// TIA Portal V18 export
FUNCTION "HMI screen" : Void   // FC18, LAD
{ S7_Optimized_Access := 'TRUE' }
VERSION : 0.1
// stored: AutoNumber true, IsIECCheckEnabled false, SetENOAutomatically false, UDAEnableTagReadback false
   VAR_TEMP
      temp1 : Bool;
      temp2 : Bool;
      temp3 : Bool;
      temp10 : Bool;
      temp11 : Bool;
      "dearing A" : Bool;
      "dearing A_1" : Bool;
      dearingA : Bool;
   END_VAR
   VAR_TEMP   // added for the SCL form of the ladder/FBD networks
      _w1 : Bool;
      _w2 : Bool;
   END_VAR
BEGIN

REGION Network 1: Metering continious screen/AD1000
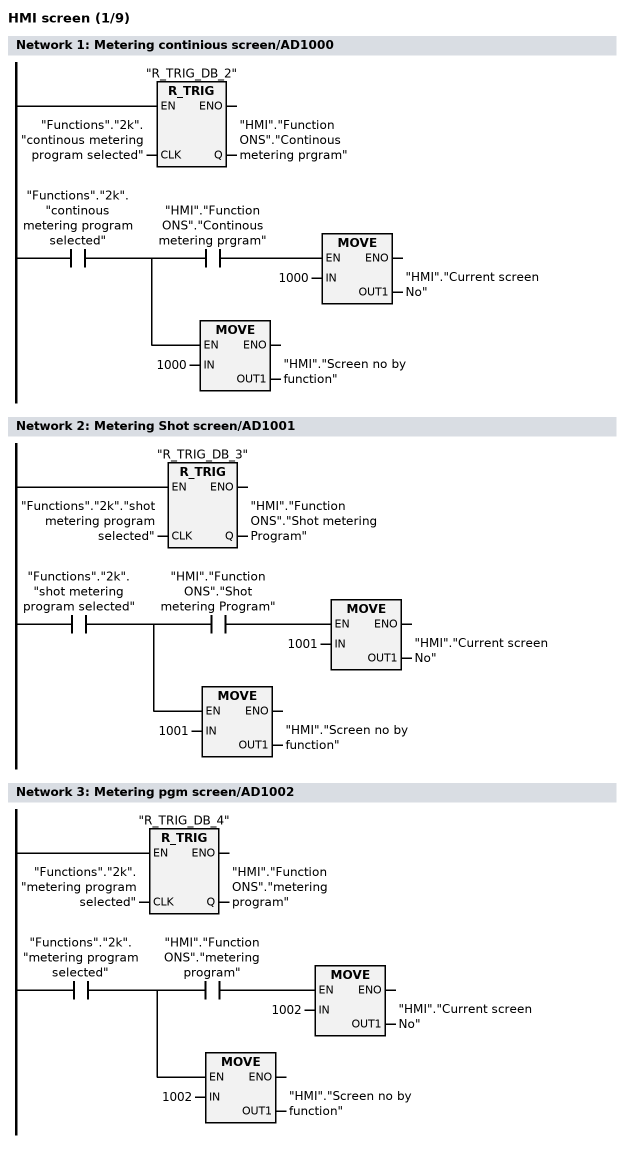
   RUNG wire#powerrail
      "R_TRIG_DB_2".R_TRIG(CLK := "Functions"."2k"."continous metering program selected", Q => "HMI"."Function ONS"."Continous metering prgram")
   END_RUNG
   RUNG wire#powerrail
      Contact( "Functions"."2k"."continous metering program selected" )
      wire#w1
      Contact( "HMI"."Function ONS"."Continous metering prgram" )
      Move(in := 1000, out1 => "HMI"."Current screen No")
   END_RUNG
   RUNG wire#w1
      Move(in := 1000, out1 => "HMI"."Screen no by function")
   END_RUNG
   // the same network as SCL:
   "R_TRIG_DB_2"(CLK := "Functions"."2k"."continous metering program selected",   // R_TRIG
                 Q => "HMI"."Function ONS"."Continous metering prgram");
   IF "Functions"."2k"."continous metering program selected" AND "HMI"."Function ONS"."Continous metering prgram" THEN
       "HMI"."Current screen No" := 1000;
   END_IF;
   IF "Functions"."2k"."continous metering program selected" THEN
       "HMI"."Screen no by function" := 1000;
   END_IF;
END_REGION

REGION Network 2: Metering Shot screen/AD1001
   RUNG wire#powerrail
      "R_TRIG_DB_3".R_TRIG(CLK := "Functions"."2k"."shot metering program selected", Q => "HMI"."Function ONS"."Shot metering Program")
   END_RUNG
   RUNG wire#powerrail
      Contact( "Functions"."2k"."shot metering program selected" )
      wire#w1
      Contact( "HMI"."Function ONS"."Shot metering Program" )
      Move(in := 1001, out1 => "HMI"."Current screen No")
   END_RUNG
   RUNG wire#w1
      Move(in := 1001, out1 => "HMI"."Screen no by function")
   END_RUNG
   // the same network as SCL:
   "R_TRIG_DB_3"(CLK := "Functions"."2k"."shot metering program selected",   // R_TRIG
                 Q => "HMI"."Function ONS"."Shot metering Program");
   IF "Functions"."2k"."shot metering program selected" AND "HMI"."Function ONS"."Shot metering Program" THEN
       "HMI"."Current screen No" := 1001;
   END_IF;
   IF "Functions"."2k"."shot metering program selected" THEN "HMI"."Screen no by function" := 1001; END_IF;
END_REGION

REGION Network 3: Metering pgm screen/AD1002
   RUNG wire#powerrail
      "R_TRIG_DB_4".R_TRIG(CLK := "Functions"."2k"."metering program selected", Q => "HMI"."Function ONS"."metering program")
   END_RUNG
   RUNG wire#powerrail
      Contact( "Functions"."2k"."metering program selected" )
      wire#w1
      Contact( "HMI"."Function ONS"."metering program" )
      Move(in := 1002, out1 => "HMI"."Current screen No")
   END_RUNG
   RUNG wire#w1
      Move(in := 1002, out1 => "HMI"."Screen no by function")
   END_RUNG
   // the same network as SCL:
   "R_TRIG_DB_4"(CLK := "Functions"."2k"."metering program selected",   // R_TRIG
                 Q => "HMI"."Function ONS"."metering program");
   IF "Functions"."2k"."metering program selected" AND "HMI"."Function ONS"."metering program" THEN
       "HMI"."Current screen No" := 1002;
   END_IF;
   IF "Functions"."2k"."metering program selected" THEN "HMI"."Screen no by function" := 1002; END_IF;
END_REGION

REGION Network 4: pre run screen/AD1003
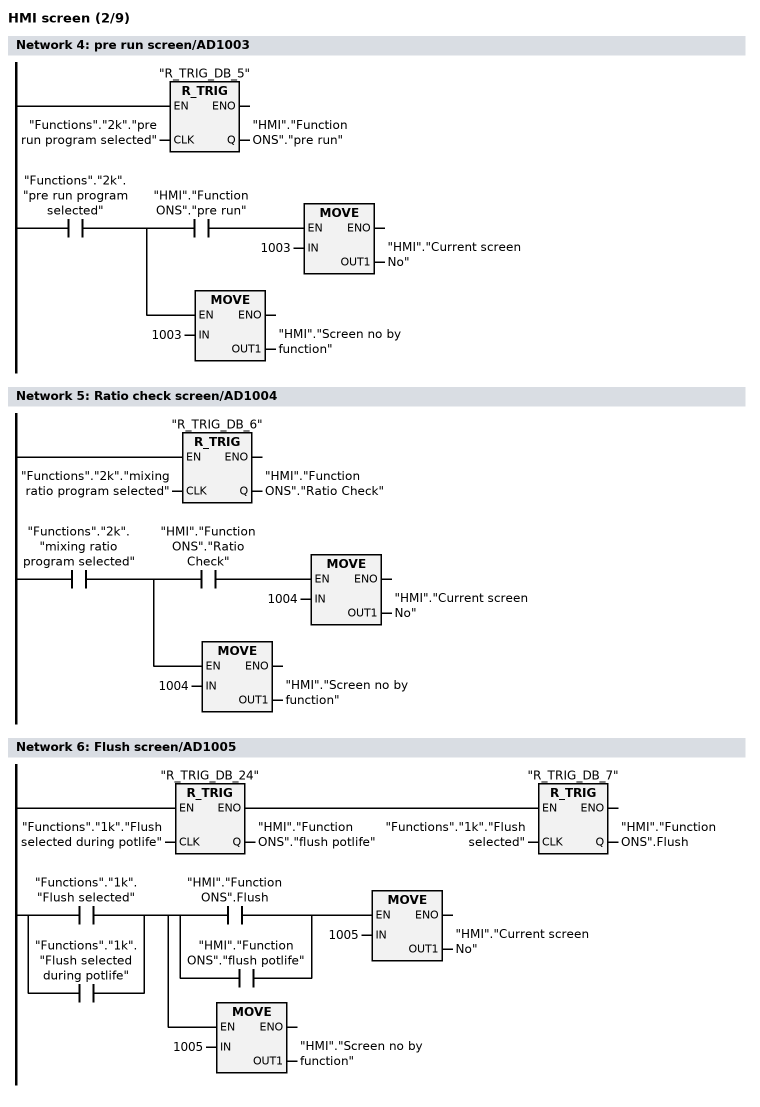
   RUNG wire#powerrail
      "R_TRIG_DB_5".R_TRIG(CLK := "Functions"."2k"."pre run program selected", Q => "HMI"."Function ONS"."pre run")
   END_RUNG
   RUNG wire#powerrail
      Contact( "Functions"."2k"."pre run program selected" )
      wire#w1
      Contact( "HMI"."Function ONS"."pre run" )
      Move(in := 1003, out1 => "HMI"."Current screen No")
   END_RUNG
   RUNG wire#w1
      Move(in := 1003, out1 => "HMI"."Screen no by function")
   END_RUNG
   // the same network as SCL:
   "R_TRIG_DB_5"(CLK := "Functions"."2k"."pre run program selected", Q => "HMI"."Function ONS"."pre run");   // R_TRIG
   IF "Functions"."2k"."pre run program selected" AND "HMI"."Function ONS"."pre run" THEN
       "HMI"."Current screen No" := 1003;
   END_IF;
   IF "Functions"."2k"."pre run program selected" THEN "HMI"."Screen no by function" := 1003; END_IF;
END_REGION

REGION Network 5: Ratio check screen/AD1004
   RUNG wire#powerrail
      "R_TRIG_DB_6".R_TRIG(CLK := "Functions"."2k"."mixing ratio program selected", Q => "HMI"."Function ONS"."Ratio Check")
   END_RUNG
   RUNG wire#powerrail
      Contact( "Functions"."2k"."mixing ratio program selected" )
      wire#w1
      Contact( "HMI"."Function ONS"."Ratio Check" )
      Move(in := 1004, out1 => "HMI"."Current screen No")
   END_RUNG
   RUNG wire#w1
      Move(in := 1004, out1 => "HMI"."Screen no by function")
   END_RUNG
   // the same network as SCL:
   "R_TRIG_DB_6"(CLK := "Functions"."2k"."mixing ratio program selected",   // R_TRIG
                 Q => "HMI"."Function ONS"."Ratio Check");
   IF "Functions"."2k"."mixing ratio program selected" AND "HMI"."Function ONS"."Ratio Check" THEN
       "HMI"."Current screen No" := 1004;
   END_IF;
   IF "Functions"."2k"."mixing ratio program selected" THEN "HMI"."Screen no by function" := 1004; END_IF;
END_REGION

REGION Network 6: Flush screen/AD1005
   RUNG wire#powerrail
      "R_TRIG_DB_24".R_TRIG(CLK := "Functions"."1k"."Flush selected during potlife", Q => "HMI"."Function ONS"."flush potlife")
      "R_TRIG_DB_7".R_TRIG(CLK := "Functions"."1k"."Flush selected", Q => "HMI"."Function ONS".Flush)
   END_RUNG
   RUNG wire#powerrail
      Contact( "Functions"."1k"."Flush selected" )
      wire#w1
      Contact( "HMI"."Function ONS".Flush )
      wire#w2
      Move(in := 1005, out1 => "HMI"."Current screen No")
   END_RUNG
   RUNG wire#powerrail
      Contact( "Functions"."1k"."Flush selected during potlife" )
   END_RUNG wire#w1
   RUNG wire#w1
      Contact( "HMI"."Function ONS"."flush potlife" )
   END_RUNG wire#w2
   RUNG wire#w1
      Move(in := 1005, out1 => "HMI"."Screen no by function")
   END_RUNG
   // the same network as SCL:
   "R_TRIG_DB_24"(CLK := "Functions"."1k"."Flush selected during potlife",   // R_TRIG
                  Q => "HMI"."Function ONS"."flush potlife",
                  ENO => #_w1);
   IF #_w1 THEN
       "R_TRIG_DB_7"(CLK := "Functions"."1k"."Flush selected", Q => "HMI"."Function ONS".Flush);   // R_TRIG
   END_IF;
   #_w2 := "Functions"."1k"."Flush selected" OR "Functions"."1k"."Flush selected during potlife";
   IF #_w2 AND ("HMI"."Function ONS".Flush OR "HMI"."Function ONS"."flush potlife") THEN
       "HMI"."Current screen No" := 1005;
   END_IF;
   IF #_w2 THEN "HMI"."Screen no by function" := 1005; END_IF;
END_REGION

REGION Network 7: dearing A screen/AD1006
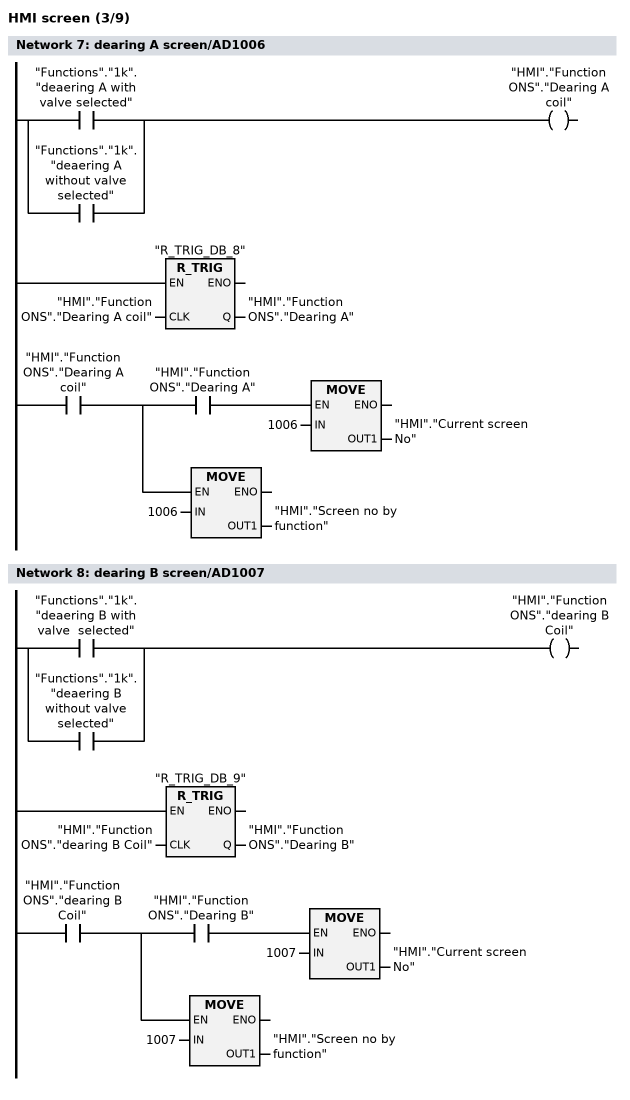
   RUNG wire#powerrail
      Contact( "Functions"."1k"."deaering A with valve selected" )
      wire#w1
      Coil( "HMI"."Function ONS"."Dearing A coil" )
   END_RUNG
   RUNG wire#powerrail
      Contact( "Functions"."1k"."deaering A without valve selected" )
   END_RUNG wire#w1
   RUNG wire#powerrail
      "R_TRIG_DB_8".R_TRIG(CLK := "HMI"."Function ONS"."Dearing A coil", Q => "HMI"."Function ONS"."Dearing A")
   END_RUNG
   RUNG wire#powerrail
      Contact( "HMI"."Function ONS"."Dearing A coil" )
      wire#w2
      Contact( "HMI"."Function ONS"."Dearing A" )
      Move(in := 1006, out1 => "HMI"."Current screen No")
   END_RUNG
   RUNG wire#w2
      Move(in := 1006, out1 => "HMI"."Screen no by function")
   END_RUNG
   // the same network as SCL:
   "HMI"."Function ONS"."Dearing A coil" := "Functions"."1k"."deaering A with valve selected" OR "Functions"."1k"."deaering A without valve selected";
   "R_TRIG_DB_8"(CLK := "HMI"."Function ONS"."Dearing A coil", Q => "HMI"."Function ONS"."Dearing A");   // R_TRIG
   IF "HMI"."Function ONS"."Dearing A coil" AND "HMI"."Function ONS"."Dearing A" THEN
       "HMI"."Current screen No" := 1006;
   END_IF;
   IF "HMI"."Function ONS"."Dearing A coil" THEN "HMI"."Screen no by function" := 1006; END_IF;
END_REGION

REGION Network 8: dearing B screen/AD1007
   RUNG wire#powerrail
      Contact( "Functions"."1k"."deaering B with valve  selected" )
      wire#w1
      Coil( "HMI"."Function ONS"."dearing B Coil" )
   END_RUNG
   RUNG wire#powerrail
      Contact( "Functions"."1k"."deaering B without valve  selected" )
   END_RUNG wire#w1
   RUNG wire#powerrail
      "R_TRIG_DB_9".R_TRIG(CLK := "HMI"."Function ONS"."dearing B Coil", Q => "HMI"."Function ONS"."Dearing B")
   END_RUNG
   RUNG wire#powerrail
      Contact( "HMI"."Function ONS"."dearing B Coil" )
      wire#w2
      Contact( "HMI"."Function ONS"."Dearing B" )
      Move(in := 1007, out1 => "HMI"."Current screen No")
   END_RUNG
   RUNG wire#w2
      Move(in := 1007, out1 => "HMI"."Screen no by function")
   END_RUNG
   // the same network as SCL:
   "HMI"."Function ONS"."dearing B Coil" := "Functions"."1k"."deaering B with valve  selected" OR "Functions"."1k"."deaering B without valve  selected";
   "R_TRIG_DB_9"(CLK := "HMI"."Function ONS"."dearing B Coil", Q => "HMI"."Function ONS"."Dearing B");   // R_TRIG
   IF "HMI"."Function ONS"."dearing B Coil" AND "HMI"."Function ONS"."Dearing B" THEN
       "HMI"."Current screen No" := 1007;
   END_IF;
   IF "HMI"."Function ONS"."dearing B Coil" THEN "HMI"."Screen no by function" := 1007; END_IF;
END_REGION

REGION Network 9: Condition Check A screen/AD1015
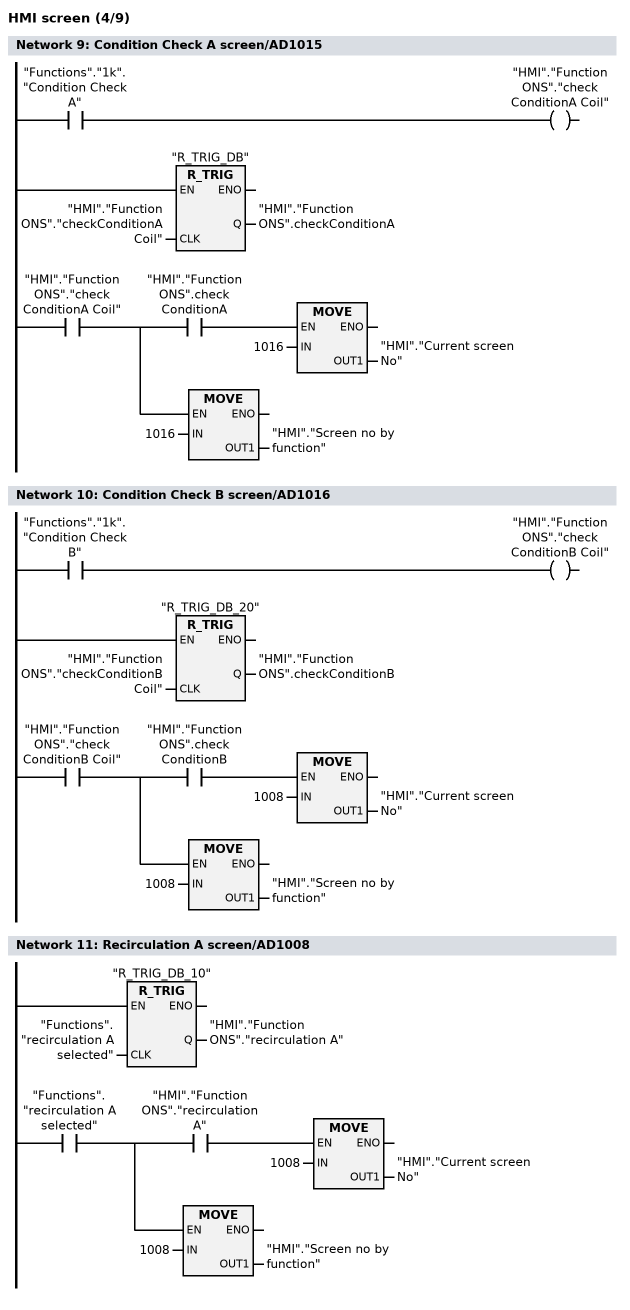
   RUNG wire#powerrail
      Contact( "Functions"."1k"."Condition Check A" )
      Coil( "HMI"."Function ONS"."checkConditionA Coil" )
   END_RUNG
   RUNG wire#powerrail
      "R_TRIG_DB".R_TRIG(CLK := "HMI"."Function ONS"."checkConditionA Coil", Q => "HMI"."Function ONS".checkConditionA)
   END_RUNG
   RUNG wire#powerrail
      Contact( "HMI"."Function ONS"."checkConditionA Coil" )
      wire#w1
      Contact( "HMI"."Function ONS".checkConditionA )
      Move(in := 1016, out1 => "HMI"."Current screen No")
   END_RUNG
   RUNG wire#w1
      Move(in := 1016, out1 => "HMI"."Screen no by function")
   END_RUNG
   // the same network as SCL:
   "HMI"."Function ONS"."checkConditionA Coil" := "Functions"."1k"."Condition Check A";
   "R_TRIG_DB"(CLK := "HMI"."Function ONS"."checkConditionA Coil", Q => "HMI"."Function ONS".checkConditionA);   // R_TRIG
   IF "HMI"."Function ONS"."checkConditionA Coil" AND "HMI"."Function ONS".checkConditionA THEN
       "HMI"."Current screen No" := 1016;
   END_IF;
   IF "HMI"."Function ONS"."checkConditionA Coil" THEN "HMI"."Screen no by function" := 1016; END_IF;
END_REGION

REGION Network 10: Condition Check B screen/AD1016
   RUNG wire#powerrail
      Contact( "Functions"."1k"."Condition Check B" )
      Coil( "HMI"."Function ONS"."checkConditionB Coil" )
   END_RUNG
   RUNG wire#powerrail
      "R_TRIG_DB_20".R_TRIG(CLK := "HMI"."Function ONS"."checkConditionB Coil", Q => "HMI"."Function ONS".checkConditionB)
   END_RUNG
   RUNG wire#powerrail
      Contact( "HMI"."Function ONS"."checkConditionB Coil" )
      wire#w1
      Contact( "HMI"."Function ONS".checkConditionB )
      Move(in := 1008, out1 => "HMI"."Current screen No")
   END_RUNG
   RUNG wire#w1
      Move(in := 1008, out1 => "HMI"."Screen no by function")
   END_RUNG
   // the same network as SCL:
   "HMI"."Function ONS"."checkConditionB Coil" := "Functions"."1k"."Condition Check B";
   "R_TRIG_DB_20"(CLK := "HMI"."Function ONS"."checkConditionB Coil", Q => "HMI"."Function ONS".checkConditionB);   // R_TRIG
   IF "HMI"."Function ONS"."checkConditionB Coil" AND "HMI"."Function ONS".checkConditionB THEN
       "HMI"."Current screen No" := 1008;
   END_IF;
   IF "HMI"."Function ONS"."checkConditionB Coil" THEN "HMI"."Screen no by function" := 1008; END_IF;
END_REGION

REGION Network 11: Recirculation A screen/AD1008
   RUNG wire#powerrail
      "R_TRIG_DB_10".R_TRIG(CLK := "Functions"."recirculation A selected", Q => "HMI"."Function ONS"."recirculation A")
   END_RUNG
   RUNG wire#powerrail
      Contact( "Functions"."recirculation A selected" )
      wire#w1
      Contact( "HMI"."Function ONS"."recirculation A" )
      Move(in := 1008, out1 => "HMI"."Current screen No")
   END_RUNG
   RUNG wire#w1
      Move(in := 1008, out1 => "HMI"."Screen no by function")
   END_RUNG
   // the same network as SCL:
   "R_TRIG_DB_10"(CLK := "Functions"."recirculation A selected", Q => "HMI"."Function ONS"."recirculation A");   // R_TRIG
   IF "Functions"."recirculation A selected" AND "HMI"."Function ONS"."recirculation A" THEN
       "HMI"."Current screen No" := 1008;
   END_IF;
   IF "Functions"."recirculation A selected" THEN "HMI"."Screen no by function" := 1008; END_IF;
END_REGION

REGION Network 12: Recirculation B screen/AD1009
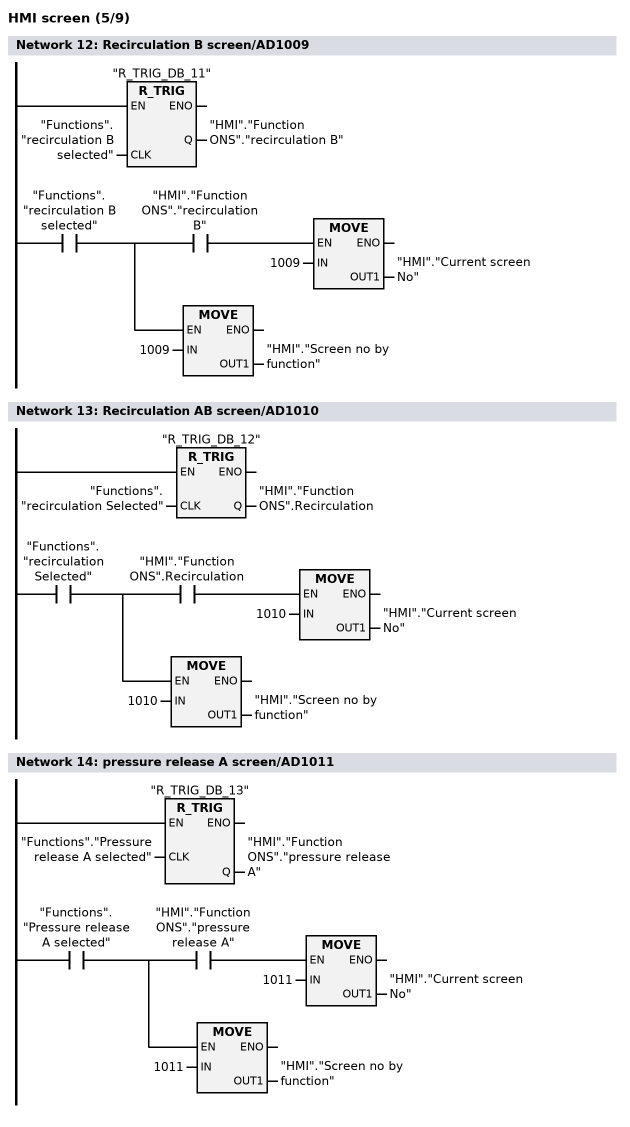
   RUNG wire#powerrail
      "R_TRIG_DB_11".R_TRIG(CLK := "Functions"."recirculation B selected", Q => "HMI"."Function ONS"."recirculation B")
   END_RUNG
   RUNG wire#powerrail
      Contact( "Functions"."recirculation B selected" )
      wire#w1
      Contact( "HMI"."Function ONS"."recirculation B" )
      Move(in := 1009, out1 => "HMI"."Current screen No")
   END_RUNG
   RUNG wire#w1
      Move(in := 1009, out1 => "HMI"."Screen no by function")
   END_RUNG
   // the same network as SCL:
   "R_TRIG_DB_11"(CLK := "Functions"."recirculation B selected", Q => "HMI"."Function ONS"."recirculation B");   // R_TRIG
   IF "Functions"."recirculation B selected" AND "HMI"."Function ONS"."recirculation B" THEN
       "HMI"."Current screen No" := 1009;
   END_IF;
   IF "Functions"."recirculation B selected" THEN "HMI"."Screen no by function" := 1009; END_IF;
END_REGION

REGION Network 13: Recirculation AB screen/AD1010
   RUNG wire#powerrail
      "R_TRIG_DB_12".R_TRIG(CLK := "Functions"."recirculation Selected", Q => "HMI"."Function ONS".Recirculation)
   END_RUNG
   RUNG wire#powerrail
      Contact( "Functions"."recirculation Selected" )
      wire#w1
      Contact( "HMI"."Function ONS".Recirculation )
      Move(in := 1010, out1 => "HMI"."Current screen No")
   END_RUNG
   RUNG wire#w1
      Move(in := 1010, out1 => "HMI"."Screen no by function")
   END_RUNG
   // the same network as SCL:
   "R_TRIG_DB_12"(CLK := "Functions"."recirculation Selected", Q => "HMI"."Function ONS".Recirculation);   // R_TRIG
   IF "Functions"."recirculation Selected" AND "HMI"."Function ONS".Recirculation THEN
       "HMI"."Current screen No" := 1010;
   END_IF;
   IF "Functions"."recirculation Selected" THEN "HMI"."Screen no by function" := 1010; END_IF;
END_REGION

REGION Network 14: pressure release A screen/AD1011
   RUNG wire#powerrail
      "R_TRIG_DB_13".R_TRIG(CLK := "Functions"."Pressure release A selected", Q => "HMI"."Function ONS"."pressure release A")
   END_RUNG
   RUNG wire#powerrail
      Contact( "Functions"."Pressure release A selected" )
      wire#w1
      Contact( "HMI"."Function ONS"."pressure release A" )
      Move(in := 1011, out1 => "HMI"."Current screen No")
   END_RUNG
   RUNG wire#w1
      Move(in := 1011, out1 => "HMI"."Screen no by function")
   END_RUNG
   // the same network as SCL:
   "R_TRIG_DB_13"(CLK := "Functions"."Pressure release A selected",   // R_TRIG
                  Q => "HMI"."Function ONS"."pressure release A");
   IF "Functions"."Pressure release A selected" AND "HMI"."Function ONS"."pressure release A" THEN
       "HMI"."Current screen No" := 1011;
   END_IF;
   IF "Functions"."Pressure release A selected" THEN "HMI"."Screen no by function" := 1011; END_IF;
END_REGION

REGION Network 15: pressure release B screen/AD1012
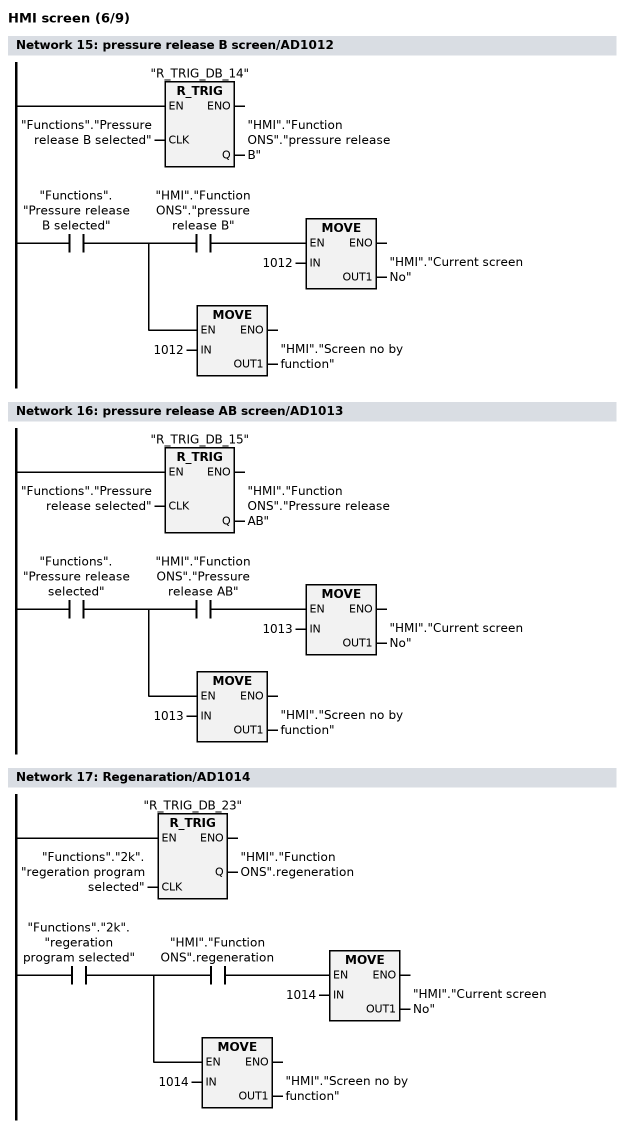
   RUNG wire#powerrail
      "R_TRIG_DB_14".R_TRIG(CLK := "Functions"."Pressure release B selected", Q => "HMI"."Function ONS"."pressure release B")
   END_RUNG
   RUNG wire#powerrail
      Contact( "Functions"."Pressure release B selected" )
      wire#w1
      Contact( "HMI"."Function ONS"."pressure release B" )
      Move(in := 1012, out1 => "HMI"."Current screen No")
   END_RUNG
   RUNG wire#w1
      Move(in := 1012, out1 => "HMI"."Screen no by function")
   END_RUNG
   // the same network as SCL:
   "R_TRIG_DB_14"(CLK := "Functions"."Pressure release B selected",   // R_TRIG
                  Q => "HMI"."Function ONS"."pressure release B");
   IF "Functions"."Pressure release B selected" AND "HMI"."Function ONS"."pressure release B" THEN
       "HMI"."Current screen No" := 1012;
   END_IF;
   IF "Functions"."Pressure release B selected" THEN "HMI"."Screen no by function" := 1012; END_IF;
END_REGION

REGION Network 16: pressure release AB screen/AD1013
   RUNG wire#powerrail
      "R_TRIG_DB_15".R_TRIG(CLK := "Functions"."Pressure release selected", Q => "HMI"."Function ONS"."Pressure release AB")
   END_RUNG
   RUNG wire#powerrail
      Contact( "Functions"."Pressure release selected" )
      wire#w1
      Contact( "HMI"."Function ONS"."Pressure release AB" )
      Move(in := 1013, out1 => "HMI"."Current screen No")
   END_RUNG
   RUNG wire#w1
      Move(in := 1013, out1 => "HMI"."Screen no by function")
   END_RUNG
   // the same network as SCL:
   "R_TRIG_DB_15"(CLK := "Functions"."Pressure release selected",   // R_TRIG
                  Q => "HMI"."Function ONS"."Pressure release AB");
   IF "Functions"."Pressure release selected" AND "HMI"."Function ONS"."Pressure release AB" THEN
       "HMI"."Current screen No" := 1013;
   END_IF;
   IF "Functions"."Pressure release selected" THEN "HMI"."Screen no by function" := 1013; END_IF;
END_REGION

REGION Network 17: Regenaration/AD1014
   RUNG wire#powerrail
      "R_TRIG_DB_23".R_TRIG(CLK := "Functions"."2k"."regeration program selected", Q => "HMI"."Function ONS".regeneration)
   END_RUNG
   RUNG wire#powerrail
      Contact( "Functions"."2k"."regeration program selected" )
      wire#w1
      Contact( "HMI"."Function ONS".regeneration )
      Move(in := 1014, out1 => "HMI"."Current screen No")
   END_RUNG
   RUNG wire#w1
      Move(in := 1014, out1 => "HMI"."Screen no by function")
   END_RUNG
   // the same network as SCL:
   "R_TRIG_DB_23"(CLK := "Functions"."2k"."regeration program selected", Q => "HMI"."Function ONS".regeneration);   // R_TRIG
   IF "Functions"."2k"."regeration program selected" AND "HMI"."Function ONS".regeneration THEN
       "HMI"."Current screen No" := 1014;
   END_IF;
   IF "Functions"."2k"."regeration program selected" THEN "HMI"."Screen no by function" := 1014; END_IF;
END_REGION

REGION Network 18: Main menu
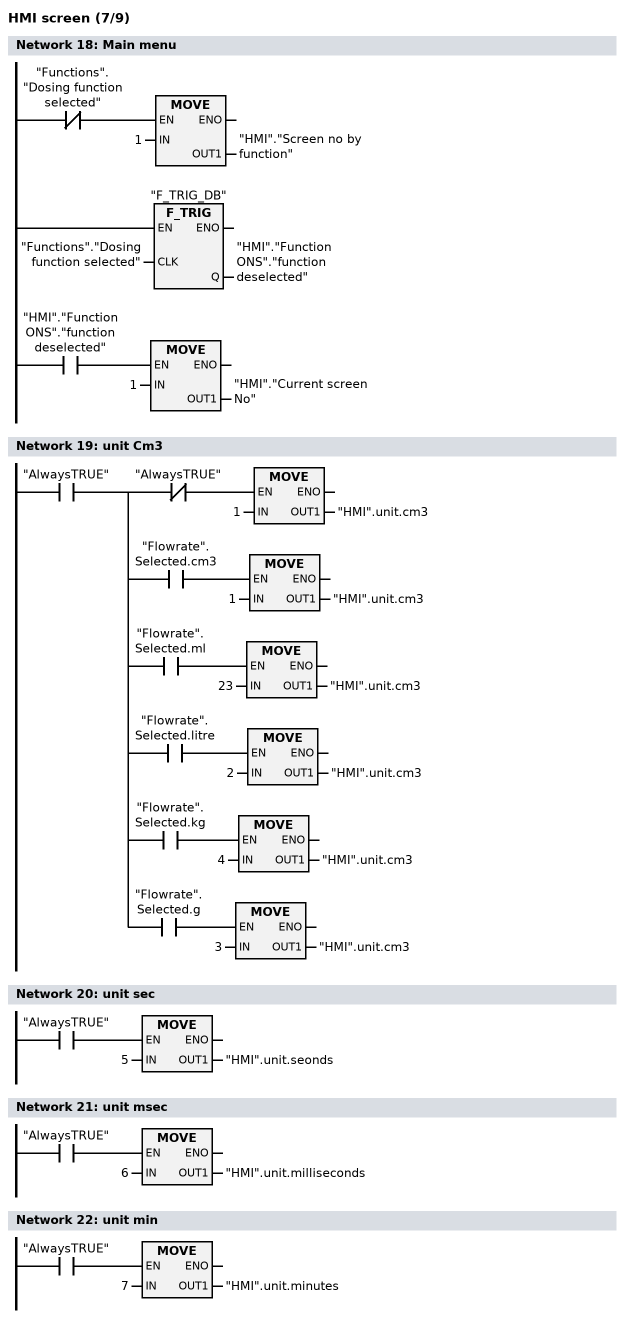
   RUNG wire#powerrail
      I_Contact( "Functions"."Dosing function selected" )
      Move(in := 1, out1 => "HMI"."Screen no by function")
   END_RUNG
   RUNG wire#powerrail
      "F_TRIG_DB".F_TRIG(CLK := "Functions"."Dosing function selected", Q => "HMI"."Function ONS"."function deselected")
   END_RUNG
   RUNG wire#powerrail
      Contact( "HMI"."Function ONS"."function deselected" )
      Move(in := 1, out1 => "HMI"."Current screen No")
   END_RUNG
   // the same network as SCL:
   IF NOT "Functions"."Dosing function selected" THEN "HMI"."Screen no by function" := 1; END_IF;
   "F_TRIG_DB"(CLK := "Functions"."Dosing function selected", Q => "HMI"."Function ONS"."function deselected");   // F_TRIG
   IF "HMI"."Function ONS"."function deselected" THEN "HMI"."Current screen No" := 1; END_IF;
END_REGION

REGION Network 19: unit Cm3
   RUNG wire#powerrail
      Contact( "AlwaysTRUE" )
      wire#w1
      I_Contact( "AlwaysTRUE" )
      Move(in := 1, out1 => "HMI".unit.cm3)
   END_RUNG
   RUNG wire#w1
      Contact( "Flowrate".Selected.cm3 )
      Move(in := 1, out1 => "HMI".unit.cm3)
   END_RUNG
   RUNG wire#w1
      Contact( "Flowrate".Selected.ml )
      Move(in := 23, out1 => "HMI".unit.cm3)
   END_RUNG
   RUNG wire#w1
      Contact( "Flowrate".Selected.litre )
      Move(in := 2, out1 => "HMI".unit.cm3)
   END_RUNG
   RUNG wire#w1
      Contact( "Flowrate".Selected.kg )
      Move(in := 4, out1 => "HMI".unit.cm3)
   END_RUNG
   RUNG wire#w1
      Contact( "Flowrate".Selected.g )
      Move(in := 3, out1 => "HMI".unit.cm3)
   END_RUNG
   // the same network as SCL:
   IF "AlwaysTRUE" AND NOT "AlwaysTRUE" THEN "HMI".unit.cm3 := 1; END_IF;
   IF "AlwaysTRUE" AND "Flowrate".Selected.cm3 THEN "HMI".unit.cm3 := 1; END_IF;
   IF "AlwaysTRUE" AND "Flowrate".Selected.ml THEN "HMI".unit.cm3 := 23; END_IF;
   IF "AlwaysTRUE" AND "Flowrate".Selected.litre THEN "HMI".unit.cm3 := 2; END_IF;
   IF "AlwaysTRUE" AND "Flowrate".Selected.kg THEN "HMI".unit.cm3 := 4; END_IF;
   IF "AlwaysTRUE" AND "Flowrate".Selected.g THEN "HMI".unit.cm3 := 3; END_IF;
END_REGION

REGION Network 20: unit sec
   RUNG wire#powerrail
      Contact( "AlwaysTRUE" )
      Move(in := 5, out1 => "HMI".unit.seonds)
   END_RUNG
   // the same network as SCL:
   IF "AlwaysTRUE" THEN "HMI".unit.seonds := 5; END_IF;
END_REGION

REGION Network 21: unit msec
   RUNG wire#powerrail
      Contact( "AlwaysTRUE" )
      Move(in := 6, out1 => "HMI".unit.milliseconds)
   END_RUNG
   // the same network as SCL:
   IF "AlwaysTRUE" THEN "HMI".unit.milliseconds := 6; END_IF;
END_REGION

REGION Network 22: unit min
   RUNG wire#powerrail
      Contact( "AlwaysTRUE" )
      Move(in := 7, out1 => "HMI".unit.minutes)
   END_RUNG
   // the same network as SCL:
   IF "AlwaysTRUE" THEN "HMI".unit.minutes := 7; END_IF;
END_REGION

REGION Network 23: unit hour
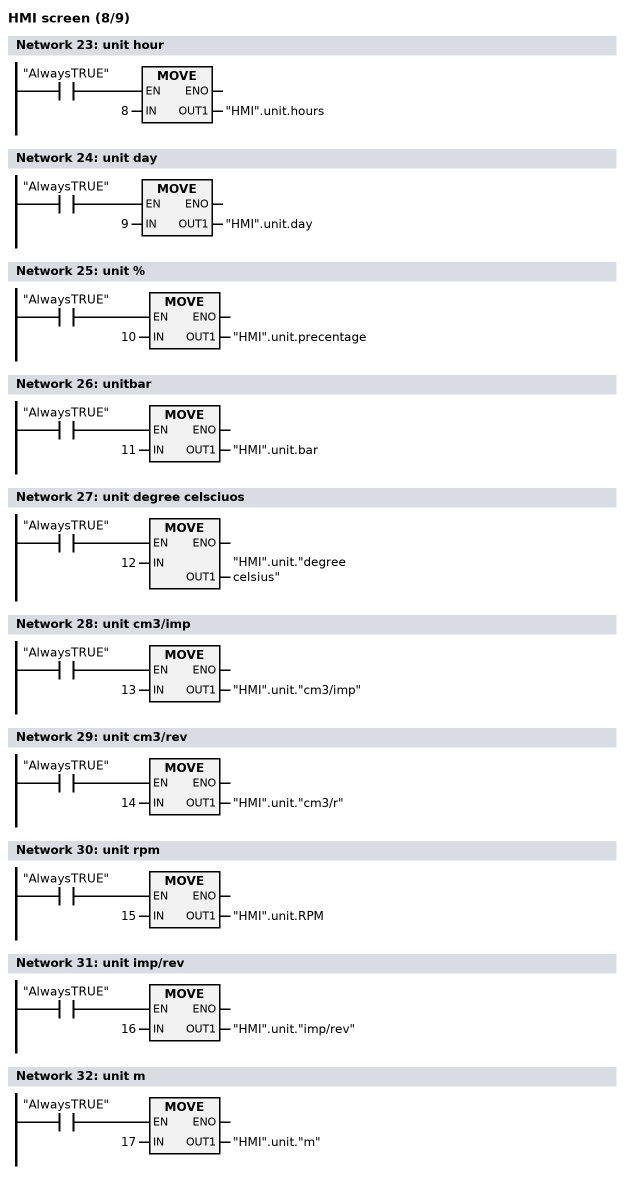
   RUNG wire#powerrail
      Contact( "AlwaysTRUE" )
      Move(in := 8, out1 => "HMI".unit.hours)
   END_RUNG
   // the same network as SCL:
   IF "AlwaysTRUE" THEN "HMI".unit.hours := 8; END_IF;
END_REGION

REGION Network 24: unit day
   RUNG wire#powerrail
      Contact( "AlwaysTRUE" )
      Move(in := 9, out1 => "HMI".unit.day)
   END_RUNG
   // the same network as SCL:
   IF "AlwaysTRUE" THEN "HMI".unit.day := 9; END_IF;
END_REGION

REGION Network 25: unit %
   RUNG wire#powerrail
      Contact( "AlwaysTRUE" )
      Move(in := 10, out1 => "HMI".unit.precentage)
   END_RUNG
   // the same network as SCL:
   IF "AlwaysTRUE" THEN "HMI".unit.precentage := 10; END_IF;
END_REGION

REGION Network 26: unitbar
   RUNG wire#powerrail
      Contact( "AlwaysTRUE" )
      Move(in := 11, out1 => "HMI".unit.bar)
   END_RUNG
   // the same network as SCL:
   IF "AlwaysTRUE" THEN "HMI".unit.bar := 11; END_IF;
END_REGION

REGION Network 27: unit degree celsciuos
   RUNG wire#powerrail
      Contact( "AlwaysTRUE" )
      Move(in := 12, out1 => "HMI".unit."degree celsius")
   END_RUNG
   // the same network as SCL:
   IF "AlwaysTRUE" THEN "HMI".unit."degree celsius" := 12; END_IF;
END_REGION

REGION Network 28: unit cm3/imp
   RUNG wire#powerrail
      Contact( "AlwaysTRUE" )
      Move(in := 13, out1 => "HMI".unit."cm3/imp")
   END_RUNG
   // the same network as SCL:
   IF "AlwaysTRUE" THEN "HMI".unit."cm3/imp" := 13; END_IF;
END_REGION

REGION Network 29: unit cm3/rev
   RUNG wire#powerrail
      Contact( "AlwaysTRUE" )
      Move(in := 14, out1 => "HMI".unit."cm3/r")
   END_RUNG
   // the same network as SCL:
   IF "AlwaysTRUE" THEN "HMI".unit."cm3/r" := 14; END_IF;
END_REGION

REGION Network 30: unit rpm
   RUNG wire#powerrail
      Contact( "AlwaysTRUE" )
      Move(in := 15, out1 => "HMI".unit.RPM)
   END_RUNG
   // the same network as SCL:
   IF "AlwaysTRUE" THEN "HMI".unit.RPM := 15; END_IF;
END_REGION

REGION Network 31: unit imp/rev
   RUNG wire#powerrail
      Contact( "AlwaysTRUE" )
      Move(in := 16, out1 => "HMI".unit."imp/rev")
   END_RUNG
   // the same network as SCL:
   IF "AlwaysTRUE" THEN "HMI".unit."imp/rev" := 16; END_IF;
END_REGION

REGION Network 32: unit m
   RUNG wire#powerrail
      Contact( "AlwaysTRUE" )
      Move(in := 17, out1 => "HMI".unit."m")
   END_RUNG
   // the same network as SCL:
   IF "AlwaysTRUE" THEN "HMI".unit."m" := 17; END_IF;
END_REGION

REGION Network 33: unit cm3/min
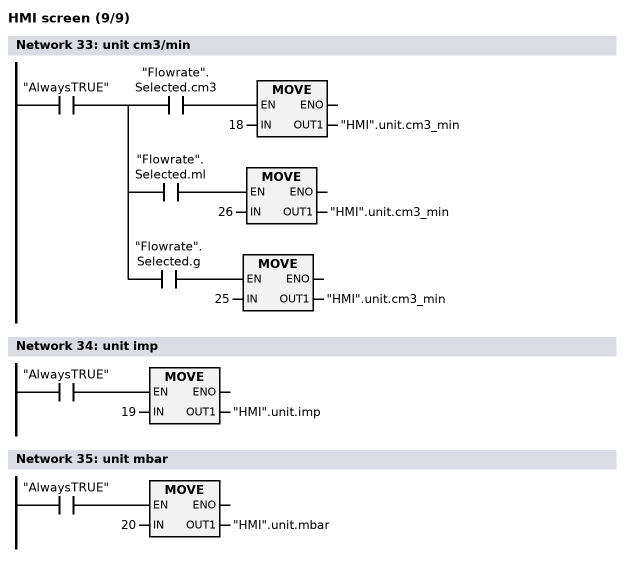
   RUNG wire#powerrail
      Contact( "AlwaysTRUE" )
      wire#w1
      Contact( "Flowrate".Selected.cm3 )
      Move(in := 18, out1 => "HMI".unit.cm3_min)
   END_RUNG
   RUNG wire#w1
      Contact( "Flowrate".Selected.ml )
      Move(in := 26, out1 => "HMI".unit.cm3_min)
   END_RUNG
   RUNG wire#w1
      Contact( "Flowrate".Selected.g )
      Move(in := 25, out1 => "HMI".unit.cm3_min)
   END_RUNG
   // the same network as SCL:
   IF "AlwaysTRUE" AND "Flowrate".Selected.cm3 THEN "HMI".unit.cm3_min := 18; END_IF;
   IF "AlwaysTRUE" AND "Flowrate".Selected.ml THEN "HMI".unit.cm3_min := 26; END_IF;
   IF "AlwaysTRUE" AND "Flowrate".Selected.g THEN "HMI".unit.cm3_min := 25; END_IF;
END_REGION

REGION Network 34: unit imp
   RUNG wire#powerrail
      Contact( "AlwaysTRUE" )
      Move(in := 19, out1 => "HMI".unit.imp)
   END_RUNG
   // the same network as SCL:
   IF "AlwaysTRUE" THEN "HMI".unit.imp := 19; END_IF;
END_REGION

REGION Network 35: unit mbar
   RUNG wire#powerrail
      Contact( "AlwaysTRUE" )
      Move(in := 20, out1 => "HMI".unit.mbar)
   END_RUNG
   // the same network as SCL:
   IF "AlwaysTRUE" THEN "HMI".unit.mbar := 20; END_IF;
END_REGION

REGION Network 36 (SCL): user logged
   IF "HMI"."HMI User" = WString#'admin' THEN
       "HMI".AdminLogged := true;

   ELSE
       "HMI".AdminLogged := false;
       "HMI".userlogged := FALSE;
   END_IF;


   IF LEN("HMI"."HMI User") > 1 THEN
       "HMI".userlogged := TRUE;
   ELSE
       "HMI".userlogged := FALSE;
   END_IF;
END_REGION

REGION Network 37 (SCL)
   "HMI"."HMI user To hmi" := "HMI"."HMI User";
END_REGION
END_FUNCTION
